(* CODESYS project ExceptionGenerator.library
   TcLibraryId: TE140x Module Vendor|ExceptionGenerator|0.0.0.3
   Company: TE140x Module Vendor
   DefaultNamespace: ExceptionGenerator
   Version: 0.0.0.3
   Placeholder: ExceptionGenerator
   Title: ExceptionGenerator

Project tree, tasks and I/O mapping:
  Version/
    global variables Global_Version
  Pous/
    function block FB_ExceptionGenerator [ST]: FB_exit, FB_init
    TcCOM Wrapper/
      function block FB_ExceptionGenerator_TcCOM_InitStruct [ST]: FB_init, FB_afterinit, Reinit, FB_exit, nTaskOid, nObjectState, ipADI, ipTcComObject, nTaskPriority, nTaskCycleTimeNs, nTaskPort, nTaskSortOrder, eTraceLevelMax, eModuleCaller, eCallerVerification, eStepSizeAdaptation, eExecutionSequence, bExecute, eAccessLockState, eInitExceptionHandling, eUpdateExceptionHandling, stModuleBuildInfo, bInitialized, stInitExceptionInfo, nCycleCount, nExceptionCount, stExeceptionInfo
  Duts/
    data type ST_FB_Main_FB_ExceptionGenerator
    data type ST_FB_exit_FB_ExceptionGenerator
    data type ST_FB_init_FB_ExceptionGenerator
    data type ST_DW_ExceptionGenerator_T
    data type ST_ExtU_ExceptionGenerator_T
    data type ST_ExtY_ExceptionGenerator_T
    data type E_ModuleCaller
    data type E_CallerVerification
    data type E_StepSizeAdaptation
    data type E_ExecutionSequence1
    data type E_FpExcptCtrlSet
    data type ST_FB_ExceptionGenerator_TcCOM_InitStruct
    data type ST_FB_init_FB_ExceptionGenerator_TcCOM_InitStruct
    data type ST_FB_afterinit_FB_ExceptionGenerator_TcCOM_InitStruct
    data type ST_Reinit_FB_ExceptionGenerator_TcCOM_InitStruct
    data type ST_FB_Main_FB_ExceptionGenerator_TcCOM_InitStruct
    data type ST_FB_exit_FB_ExceptionGenerator_TcCOM_InitStruct
    data type ST_GetnTaskOid_FB_ExceptionGenerator_TcCOM_InitStruct
    data type ST_SetnTaskOid_FB_ExceptionGenerator_TcCOM_InitStruct
    data type ST_GetnObjectState_FB_ExceptionGenerator_TcCOM_InitStruct
    data type ST_SetnObjectState_FB_ExceptionGenerator_TcCOM_InitStruct
    data type ST_GetipADI_FB_ExceptionGenerator_TcCOM_InitStruct
    data type ST_SetipADI_FB_ExceptionGenerator_TcCOM_InitStruct
    data type ST_GetipTcComObject_FB_ExceptionGenerator_TcCOM_InitStruct
    data type ST_SetipTcComObject_FB_ExceptionGenerator_TcCOM_InitStruct
    data type ST_ExceptionInfo
    data type ST_ExecutionInfo
    data type ST_GetnTaskPriority_FB_ExceptionGenerator_TcCOM_InitStruct
    data type ST_SetnTaskPriority_FB_ExceptionGenerator_TcCOM_InitStruct
    data type ST_GetnTaskCycleTimeNs_FB_ExceptionGenerator_TcCOM_InitStruct
    data type ST_SetnTaskCycleTimeNs_FB_ExceptionGenerator_TcCOM_InitStruct
    data type ST_GetnTaskPort_FB_ExceptionGenerator_TcCOM_InitStruct
    data type ST_SetnTaskPort_FB_ExceptionGenerator_TcCOM_InitStruct
    data type ST_GetnTaskSortOrder_FB_ExceptionGenerator_TcCOM_InitStruct
    data type ST_SetnTaskSortOrder_FB_ExceptionGenerator_TcCOM_InitStruct
    data type ST_GeteTraceLevelMax_FB_ExceptionGenerator_TcCOM_InitStruct
    data type ST_SeteTraceLevelMax_FB_ExceptionGenerator_TcCOM_InitStruct
    data type ST_GeteModuleCaller_FB_ExceptionGenerator_TcCOM_InitStruct
    data type ST_SeteModuleCaller_FB_ExceptionGenerator_TcCOM_InitStruct
    data type ST_GeteCallerVerification_FB_ExceptionGenerator_TcCOM_InitStruct
    data type ST_SeteCallerVerification_FB_ExceptionGenerator_TcCOM_InitStruct
    data type ST_GeteStepSizeAdaptation_FB_ExceptionGenerator_TcCOM_InitStruct
    data type ST_SeteStepSizeAdaptation_FB_ExceptionGenerator_TcCOM_InitStruct
    data type ST_GeteExecutionSequence_FB_ExceptionGenerator_TcCOM_InitStruct
    data type ST_SeteExecutionSequence_FB_ExceptionGenerator_TcCOM_InitStruct
    data type ST_GetbExecute_FB_ExceptionGenerator_TcCOM_InitStruct
    data type ST_SetbExecute_FB_ExceptionGenerator_TcCOM_InitStruct
    data type ST_GeteAccessLockState_FB_ExceptionGenerator_TcCOM_InitStruct
    data type ST_SeteAccessLockState_FB_ExceptionGenerator_TcCOM_InitStruct
    data type ST_GeteInitExceptionHandling_FB_ExceptionGenerator_TcCOM_InitStruct
    data type ST_SeteInitExceptionHandling_FB_ExceptionGenerator_TcCOM_InitStruct
    data type ST_GeteUpdateExceptionHandling_FB_ExceptionGenerator_TcCOM_InitStruct
    data type ST_SeteUpdateExceptionHandling_FB_ExceptionGenerator_TcCOM_InitStruct
    data type ST_ModuleBuildInfo
    data type ST_GetstModuleBuildInfo_FB_ExceptionGenerator_TcCOM_InitStruct
    data type ST_SetstModuleBuildInfo_FB_ExceptionGenerator_TcCOM_InitStruct
    data type ST_GetbInitialized_FB_ExceptionGenerator_TcCOM_InitStruct
    data type ST_SetbInitialized_FB_ExceptionGenerator_TcCOM_InitStruct
    data type ST_GetstInitExceptionInfo_FB_ExceptionGenerator_TcCOM_InitStruct
    data type ST_SetstInitExceptionInfo_FB_ExceptionGenerator_TcCOM_InitStruct
    data type ST_GetnCycleCount_FB_ExceptionGenerator_TcCOM_InitStruct
    data type ST_SetnCycleCount_FB_ExceptionGenerator_TcCOM_InitStruct
    data type ST_GetnExceptionCount_FB_ExceptionGenerator_TcCOM_InitStruct
    data type ST_SetnExceptionCount_FB_ExceptionGenerator_TcCOM_InitStruct
    data type ST_GetstExeceptionInfo_FB_ExceptionGenerator_TcCOM_InitStruct
    data type ST_SetstExeceptionInfo_FB_ExceptionGenerator_TcCOM_InitStruct
*)

// Duts/ST_FB_Main_FB_ExceptionGenerator

	{attribute 'TcIecLibraryType'}
{attribute 'hide'}
TYPE ST_FB_Main_FB_ExceptionGenerator : 
	STRUCT
		 {attribute 'GUID' := '18071995-0000-0000-0000-000000000018'}
		pInst : PVOID;
		result : BOOL;
		 {attribute 'hide'}
		_reserved1 : UINT_24_56;
	END_STRUCT
END_TYPE

// Duts/ST_FB_exit_FB_ExceptionGenerator

	{attribute 'TcIecLibraryType'}
{attribute 'hide'}
TYPE ST_FB_exit_FB_ExceptionGenerator : 
	STRUCT
		 {attribute 'GUID' := '18071995-0000-0000-0000-000000000018'}
		pInst : PVOID;
		bInCopyCode : BOOL;
		result : BOOL;
		 {attribute 'hide'}
		_reserved1 : UINT_16_48;
	END_STRUCT
END_TYPE

// Duts/ST_FB_init_FB_ExceptionGenerator

	{attribute 'TcIecLibraryType'}
{attribute 'hide'}
TYPE ST_FB_init_FB_ExceptionGenerator : 
	STRUCT
		 {attribute 'GUID' := '18071995-0000-0000-0000-000000000018'}
		pInst : PVOID;
		bInitRetains : BOOL;
		bInCopyCode : BOOL;
		result : BOOL;
		 {attribute 'hide'}
		_reserved1 : UINT_8_40;
	END_STRUCT
END_TYPE

// Duts/ST_DW_ExceptionGenerator_T

	{attribute 'TcIecLibraryType'}
TYPE ST_DW_ExceptionGenerator_T : 
	STRUCT
		fCounter : LREAL;
		fa : LREAL;
		fb : LREAL;
		ffPosInf : LREAL;
		ffNegInf : LREAL;
	END_STRUCT
END_TYPE

// Duts/ST_ExtU_ExceptionGenerator_T

	{attribute 'TcIecLibraryType'}
TYPE ST_ExtU_ExceptionGenerator_T : 
	STRUCT
		bDivByZero : BOOL;
		bFloatingPoint : BOOL;
	END_STRUCT
END_TYPE

// Duts/ST_ExtY_ExceptionGenerator_T

	{attribute 'TcIecLibraryType'}
TYPE ST_ExtY_ExceptionGenerator_T : 
	STRUCT
		fResult : LREAL;
		fCounter : LREAL;
	END_STRUCT
END_TYPE

// Duts/E_ModuleCaller

	{attribute 'TcIecLibraryType'}
TYPE E_ModuleCaller : (
	CyclicTask:=0, 	(* Add to the specified cyclic caller tasks. *)
	Module:=1	(* Don't add to cyclic callers. The module can be called from other TwinCAT modules (e. g. a PLC). *)
) DINT;
END_TYPE

// Duts/E_CallerVerification

	{attribute 'TcIecLibraryType'}
TYPE E_CallerVerification : (
	Default:=0, 	(* Verify the caller task only if the "ModuleCaller" parameter is set to "Module" but not when added to cyclic caller tasks. *)
	Always:=1, 	(* Always verify the caller context to prevent concurrent execution of model code and corresponding DataArea mappings. *)
	Never:=2	(* Skip caller verification to reduce execution times. *)
) DINT;
END_TYPE

// Duts/E_StepSizeAdaptation

	{attribute 'TcIecLibraryType'}
TYPE E_StepSizeAdaptation : (
	RequireMatchingTaskCycleTime:=0, 	(* Don't accept task cycle times other than the Simulink step sizes. *)
	UseTaskCycleTime:=1, 	(* Adapt the Smulink step sizes to the task cycle times. *)
	UseModelStepSize:=2	(* Keep the Smulink step sizes, independent of the callers cycle time. *)
) DINT;
END_TYPE

// Duts/E_ExecutionSequence1

	{attribute 'TcIecLibraryType'}
TYPE E_ExecutionSequence1 : (
	UpdateBeforeOutputMapping:=0, 	(* Input mapping -> State and output update -> Output mapping -> ADS processing *)
	IoAtTaskBegin:=1	(* Input mapping -> Code execution -> Output update -> ADS processing *)
) DINT;
END_TYPE

// Duts/E_FpExcptCtrlSet

	{attribute 'TcIecLibraryType'}
TYPE E_FpExcptCtrlSet : (
	CallerExceptions:=1, 	(* Use the floating point exception settings provided by the caller *)
	ThrowExceptions:=3, 	(* Enable floating point exceptions on invalid operations and divisions by zero *)
	SuppressExceptions:=12, 	(* Disable floating point exceptions. *)
	LogExceptions:=19, 	(* Log exception information. *)
	LogAndHold:=51, 	(* Log exception information and puase execution of the cyclic code after completion of the actual cycle *)
	LogAndCatch:=83, 	(* Log exception information and immediately terminate execution of the cyclic code. Reinitialization is required to restart. *)
	LogAndDump:=147, 	(* Log exception information, create a dump file with detailed exception information and try to continue execution of the cyclic code *)
	LogHoldAndDump:=179, 	(* Log exception information, create a dump file with detailed exception information and puase execution of the cyclic code after completion of the actual cycle *)
	LogCatchAndDump:=211	(* Log exception information, create a dump file with detailed exception information and immediately terminate execution of the cyclic code. Reinitialization is required to restart. *)
) USINT;
END_TYPE

// Duts/ST_FB_ExceptionGenerator_TcCOM_InitStruct

	{attribute 'TcIecLibraryType'}
TYPE ST_FB_ExceptionGenerator_TcCOM_InitStruct : 
	STRUCT
		 {attribute 'GUID' := '18071995-0000-0000-0000-000000000061'}
		eObjState : TCOM_STATE := TCOM_STATE.TCOM_STATE_OP;
		 {attribute 'GUID' := '18071995-0000-0000-0000-00000000000F'}
		nOid : OTCID := 4294967295;
		 {attribute 'GUID' := '18071995-0000-0000-0000-00000000000F'}
		nTaskOid : OTCID;
		{attribute 'hide'}
		nTaskPriority : UDINT;
		{attribute 'hide'}
		nTaskCycleTimeNs : UDINT;
		{attribute 'hide'}
		nTaskPort : UINT;
		 {attribute 'hide'}
		_reserved1 : UINT;
		nTaskSortOrder : UDINT;
		 {attribute 'GUID' := '8007AE3B-86BB-40F2-B385-EF87FCC239A4'}
		eTraceLevelMax : TcTraceLevel := TcTraceLevel.tlInfo;
		eModuleCaller : E_ModuleCaller := E_ModuleCaller.CyclicTask;
		eCallerVerification : E_CallerVerification := E_CallerVerification.Default;
		eStepSizeAdaptation : E_StepSizeAdaptation := E_StepSizeAdaptation.RequireMatchingTaskCycleTime;
		eExecutionSequence : E_ExecutionSequence1 := E_ExecutionSequence1.UpdateBeforeOutputMapping;
		bExecute : BOOL := TRUE;
		 {attribute 'hide'}
		_reserved2 : ARRAY [1..3] OF USINT;
		 {attribute 'GUID' := '18071995-0000-0000-0000-000000000061'}
		eAccessLockState : TCOM_STATE := TCOM_STATE.TCOM_STATE_OP;
		eInitExceptionHandling : E_FpExcptCtrlSet := E_FpExcptCtrlSet.LogCatchAndDump;
		eUpdateExceptionHandling : E_FpExcptCtrlSet := E_FpExcptCtrlSet.LogCatchAndDump;
		 {attribute 'hide'}
		_reserved3 : UINT;
	END_STRUCT
END_TYPE

// Duts/ST_FB_init_FB_ExceptionGenerator_TcCOM_InitStruct

	{attribute 'TcIecLibraryType'}
{attribute 'hide'}
TYPE ST_FB_init_FB_ExceptionGenerator_TcCOM_InitStruct : 
	STRUCT
		 {attribute 'GUID' := '18071995-0000-0000-0000-000000000018'}
		pInst : PVOID;
		bInitRetains : BOOL;
		bInCopyCode : BOOL;
		 {attribute 'hide'}
		_reserved1 : UINT;
		stInit : ST_FB_ExceptionGenerator_TcCOM_InitStruct;
		result : BOOL;
		 {attribute 'hide'}
		_reserved2 : UINT_24_56;
	END_STRUCT
END_TYPE

// Duts/ST_FB_afterinit_FB_ExceptionGenerator_TcCOM_InitStruct

	{attribute 'TcIecLibraryType'}
{attribute 'hide'}
TYPE ST_FB_afterinit_FB_ExceptionGenerator_TcCOM_InitStruct : 
	STRUCT
		 {attribute 'GUID' := '18071995-0000-0000-0000-000000000018'}
		pInst : PVOID;
		result : BOOL;
		 {attribute 'hide'}
		_reserved1 : UINT_24_56;
	END_STRUCT
END_TYPE

// Duts/ST_Reinit_FB_ExceptionGenerator_TcCOM_InitStruct

	{attribute 'TcIecLibraryType'}
{attribute 'hide'}
TYPE ST_Reinit_FB_ExceptionGenerator_TcCOM_InitStruct : 
	STRUCT
		 {attribute 'GUID' := '18071995-0000-0000-0000-000000000018'}
		pInst : PVOID;
		stReInit : ST_FB_ExceptionGenerator_TcCOM_InitStruct;
		result : BOOL;
		 {attribute 'hide'}
		_reserved1 : ARRAY [1..3] OF USINT;
	END_STRUCT
END_TYPE

// Duts/ST_FB_Main_FB_ExceptionGenerator_TcCOM_InitStruct

	{attribute 'TcIecLibraryType'}
{attribute 'hide'}
TYPE ST_FB_Main_FB_ExceptionGenerator_TcCOM_InitStruct : 
	STRUCT
		 {attribute 'GUID' := '18071995-0000-0000-0000-000000000018'}
		pInst : PVOID;
		result : BOOL;
		 {attribute 'hide'}
		_reserved1 : UINT_24_56;
	END_STRUCT
END_TYPE

// Duts/ST_FB_exit_FB_ExceptionGenerator_TcCOM_InitStruct

	{attribute 'TcIecLibraryType'}
{attribute 'hide'}
TYPE ST_FB_exit_FB_ExceptionGenerator_TcCOM_InitStruct : 
	STRUCT
		 {attribute 'GUID' := '18071995-0000-0000-0000-000000000018'}
		pInst : PVOID;
		bInCopyCode : BOOL;
		result : BOOL;
		 {attribute 'hide'}
		_reserved1 : UINT_16_48;
	END_STRUCT
END_TYPE

// Duts/ST_GetnTaskOid_FB_ExceptionGenerator_TcCOM_InitStruct

	{attribute 'TcIecLibraryType'}
{attribute 'hide'}
TYPE ST_GetnTaskOid_FB_ExceptionGenerator_TcCOM_InitStruct : 
	STRUCT
		 {attribute 'GUID' := '18071995-0000-0000-0000-000000000018'}
		pInst : PVOID;
		result : UDINT;
		 {attribute 'hide'}
		_reserved1 : UINT_0_32;
	END_STRUCT
END_TYPE

// Duts/ST_SetnTaskOid_FB_ExceptionGenerator_TcCOM_InitStruct

	{attribute 'TcIecLibraryType'}
{attribute 'hide'}
TYPE ST_SetnTaskOid_FB_ExceptionGenerator_TcCOM_InitStruct : 
	STRUCT
		 {attribute 'GUID' := '18071995-0000-0000-0000-000000000018'}
		pInst : PVOID;
		nParam : UDINT;
		 {attribute 'hide'}
		_reserved1 : UINT_0_32;
	END_STRUCT
END_TYPE

// Duts/ST_GetnObjectState_FB_ExceptionGenerator_TcCOM_InitStruct

	{attribute 'TcIecLibraryType'}
{attribute 'hide'}
TYPE ST_GetnObjectState_FB_ExceptionGenerator_TcCOM_InitStruct : 
	STRUCT
		 {attribute 'GUID' := '18071995-0000-0000-0000-000000000018'}
		pInst : PVOID;
		 {attribute 'GUID' := '18071995-0000-0000-0000-000000000061'}
		result : TCOM_STATE;
		 {attribute 'hide'}
		_reserved1 : UINT_0_32;
	END_STRUCT
END_TYPE

// Duts/ST_SetnObjectState_FB_ExceptionGenerator_TcCOM_InitStruct

	{attribute 'TcIecLibraryType'}
{attribute 'hide'}
TYPE ST_SetnObjectState_FB_ExceptionGenerator_TcCOM_InitStruct : 
	STRUCT
		 {attribute 'GUID' := '18071995-0000-0000-0000-000000000018'}
		pInst : PVOID;
		 {attribute 'GUID' := '18071995-0000-0000-0000-000000000061'}
		eParam : TCOM_STATE;
		 {attribute 'hide'}
		_reserved1 : UINT_0_32;
	END_STRUCT
END_TYPE

// Duts/ST_GetipADI_FB_ExceptionGenerator_TcCOM_InitStruct

	{attribute 'TcIecLibraryType'}
{attribute 'hide'}
TYPE ST_GetipADI_FB_ExceptionGenerator_TcCOM_InitStruct : 
	STRUCT
		 {attribute 'GUID' := '18071995-0000-0000-0000-000000000018'}
		pInst : PVOID;
		 {attribute 'GUID' := '03000012-0000-0000-E000-000000000064'}
		result : ITcADI;
	END_STRUCT
END_TYPE

// Duts/ST_SetipADI_FB_ExceptionGenerator_TcCOM_InitStruct

	{attribute 'TcIecLibraryType'}
{attribute 'hide'}
TYPE ST_SetipADI_FB_ExceptionGenerator_TcCOM_InitStruct : 
	STRUCT
		 {attribute 'GUID' := '18071995-0000-0000-0000-000000000018'}
		pInst : PVOID;
		 {attribute 'GUID' := '03000012-0000-0000-E000-000000000064'}
		ipParam : ITcADI;
	END_STRUCT
END_TYPE

// Duts/ST_GetipTcComObject_FB_ExceptionGenerator_TcCOM_InitStruct

	{attribute 'TcIecLibraryType'}
{attribute 'hide'}
TYPE ST_GetipTcComObject_FB_ExceptionGenerator_TcCOM_InitStruct : 
	STRUCT
		 {attribute 'GUID' := '18071995-0000-0000-0000-000000000018'}
		pInst : PVOID;
		 {attribute 'GUID' := '00000012-0000-0000-E000-000000000064'}
		result : ITComObject;
	END_STRUCT
END_TYPE

// Duts/ST_SetipTcComObject_FB_ExceptionGenerator_TcCOM_InitStruct

	{attribute 'TcIecLibraryType'}
{attribute 'hide'}
TYPE ST_SetipTcComObject_FB_ExceptionGenerator_TcCOM_InitStruct : 
	STRUCT
		 {attribute 'GUID' := '18071995-0000-0000-0000-000000000018'}
		pInst : PVOID;
		 {attribute 'GUID' := '00000012-0000-0000-E000-000000000064'}
		ipParam : ITComObject;
	END_STRUCT
END_TYPE

// Duts/ST_ExceptionInfo

	{attribute 'TcIecLibraryType'}
TYPE ST_ExceptionInfo : 
	STRUCT
		nExceptionCode : DINT;
		 {attribute 'GUID' := '18071995-0000-0000-0000-00010000007F'}
		sTmxName : STRING(127);
		nTmxVersion : UDINT;
		 {attribute 'hide'}
		_reserved1 : ARRAY [1..12] OF USINT;
		nInstructionAddr : UDINT;
		nReturnAddr : UDINT;
		 {attribute 'hide'}
		_reserved2 : ARRAY [1..12] OF USINT;
		bDumpCreated : BOOL;
		 {attribute 'hide'}
		_reserved3 : ARRAY [1..3] OF USINT;
	END_STRUCT
END_TYPE

// Duts/ST_ExecutionInfo

	{attribute 'TcIecLibraryType'}
{attribute 'pack_mode' := '1'}
TYPE ST_ExecutionInfo : 
	STRUCT
		nCycleCount : ULINT;
		nExceptionCount : ULINT;
		stActException : ST_ExceptionInfo;
	END_STRUCT
END_TYPE

// Duts/ST_GetnTaskPriority_FB_ExceptionGenerator_TcCOM_InitStruct

	{attribute 'TcIecLibraryType'}
{attribute 'hide'}
TYPE ST_GetnTaskPriority_FB_ExceptionGenerator_TcCOM_InitStruct : 
	STRUCT
		 {attribute 'GUID' := '18071995-0000-0000-0000-000000000018'}
		pInst : PVOID;
		result : UDINT;
		 {attribute 'hide'}
		_reserved1 : UINT_0_32;
	END_STRUCT
END_TYPE

// Duts/ST_SetnTaskPriority_FB_ExceptionGenerator_TcCOM_InitStruct

	{attribute 'TcIecLibraryType'}
{attribute 'hide'}
TYPE ST_SetnTaskPriority_FB_ExceptionGenerator_TcCOM_InitStruct : 
	STRUCT
		 {attribute 'GUID' := '18071995-0000-0000-0000-000000000018'}
		pInst : PVOID;
		nParam : UDINT;
		 {attribute 'hide'}
		_reserved1 : UINT_0_32;
	END_STRUCT
END_TYPE

// Duts/ST_GetnTaskCycleTimeNs_FB_ExceptionGenerator_TcCOM_InitStruct

	{attribute 'TcIecLibraryType'}
{attribute 'hide'}
TYPE ST_GetnTaskCycleTimeNs_FB_ExceptionGenerator_TcCOM_InitStruct : 
	STRUCT
		 {attribute 'GUID' := '18071995-0000-0000-0000-000000000018'}
		pInst : PVOID;
		result : UDINT;
		 {attribute 'hide'}
		_reserved1 : UINT_0_32;
	END_STRUCT
END_TYPE

// Duts/ST_SetnTaskCycleTimeNs_FB_ExceptionGenerator_TcCOM_InitStruct

	{attribute 'TcIecLibraryType'}
{attribute 'hide'}
TYPE ST_SetnTaskCycleTimeNs_FB_ExceptionGenerator_TcCOM_InitStruct : 
	STRUCT
		 {attribute 'GUID' := '18071995-0000-0000-0000-000000000018'}
		pInst : PVOID;
		nParam : UDINT;
		 {attribute 'hide'}
		_reserved1 : UINT_0_32;
	END_STRUCT
END_TYPE

// Duts/ST_GetnTaskPort_FB_ExceptionGenerator_TcCOM_InitStruct

	{attribute 'TcIecLibraryType'}
{attribute 'hide'}
TYPE ST_GetnTaskPort_FB_ExceptionGenerator_TcCOM_InitStruct : 
	STRUCT
		 {attribute 'GUID' := '18071995-0000-0000-0000-000000000018'}
		pInst : PVOID;
		result : UINT;
		 {attribute 'hide'}
		_reserved1 : UINT_16_48;
	END_STRUCT
END_TYPE

// Duts/ST_SetnTaskPort_FB_ExceptionGenerator_TcCOM_InitStruct

	{attribute 'TcIecLibraryType'}
{attribute 'hide'}
TYPE ST_SetnTaskPort_FB_ExceptionGenerator_TcCOM_InitStruct : 
	STRUCT
		 {attribute 'GUID' := '18071995-0000-0000-0000-000000000018'}
		pInst : PVOID;
		nParam : UINT;
		 {attribute 'hide'}
		_reserved1 : UINT_16_48;
	END_STRUCT
END_TYPE

// Duts/ST_GetnTaskSortOrder_FB_ExceptionGenerator_TcCOM_InitStruct

	{attribute 'TcIecLibraryType'}
{attribute 'hide'}
TYPE ST_GetnTaskSortOrder_FB_ExceptionGenerator_TcCOM_InitStruct : 
	STRUCT
		 {attribute 'GUID' := '18071995-0000-0000-0000-000000000018'}
		pInst : PVOID;
		result : UDINT;
		 {attribute 'hide'}
		_reserved1 : UINT_0_32;
	END_STRUCT
END_TYPE

// Duts/ST_SetnTaskSortOrder_FB_ExceptionGenerator_TcCOM_InitStruct

	{attribute 'TcIecLibraryType'}
{attribute 'hide'}
TYPE ST_SetnTaskSortOrder_FB_ExceptionGenerator_TcCOM_InitStruct : 
	STRUCT
		 {attribute 'GUID' := '18071995-0000-0000-0000-000000000018'}
		pInst : PVOID;
		nParam : UDINT;
		 {attribute 'hide'}
		_reserved1 : UINT_0_32;
	END_STRUCT
END_TYPE

// Duts/ST_GeteTraceLevelMax_FB_ExceptionGenerator_TcCOM_InitStruct

	{attribute 'TcIecLibraryType'}
{attribute 'hide'}
TYPE ST_GeteTraceLevelMax_FB_ExceptionGenerator_TcCOM_InitStruct : 
	STRUCT
		 {attribute 'GUID' := '18071995-0000-0000-0000-000000000018'}
		pInst : PVOID;
		 {attribute 'GUID' := '8007AE3B-86BB-40F2-B385-EF87FCC239A4'}
		result : TcTraceLevel;
		 {attribute 'hide'}
		_reserved1 : UINT_0_32;
	END_STRUCT
END_TYPE

// Duts/ST_SeteTraceLevelMax_FB_ExceptionGenerator_TcCOM_InitStruct

	{attribute 'TcIecLibraryType'}
{attribute 'hide'}
TYPE ST_SeteTraceLevelMax_FB_ExceptionGenerator_TcCOM_InitStruct : 
	STRUCT
		 {attribute 'GUID' := '18071995-0000-0000-0000-000000000018'}
		pInst : PVOID;
		 {attribute 'GUID' := '8007AE3B-86BB-40F2-B385-EF87FCC239A4'}
		eParam : TcTraceLevel;
		 {attribute 'hide'}
		_reserved1 : UINT_0_32;
	END_STRUCT
END_TYPE

// Duts/ST_GeteModuleCaller_FB_ExceptionGenerator_TcCOM_InitStruct

	{attribute 'TcIecLibraryType'}
{attribute 'hide'}
TYPE ST_GeteModuleCaller_FB_ExceptionGenerator_TcCOM_InitStruct : 
	STRUCT
		 {attribute 'GUID' := '18071995-0000-0000-0000-000000000018'}
		pInst : PVOID;
		result : E_ModuleCaller;
		 {attribute 'hide'}
		_reserved1 : UINT_0_32;
	END_STRUCT
END_TYPE

// Duts/ST_SeteModuleCaller_FB_ExceptionGenerator_TcCOM_InitStruct

	{attribute 'TcIecLibraryType'}
{attribute 'hide'}
TYPE ST_SeteModuleCaller_FB_ExceptionGenerator_TcCOM_InitStruct : 
	STRUCT
		 {attribute 'GUID' := '18071995-0000-0000-0000-000000000018'}
		pInst : PVOID;
		eParam : E_ModuleCaller;
		 {attribute 'hide'}
		_reserved1 : UINT_0_32;
	END_STRUCT
END_TYPE

// Duts/ST_GeteCallerVerification_FB_ExceptionGenerator_TcCOM_InitStruct

	{attribute 'TcIecLibraryType'}
{attribute 'hide'}
TYPE ST_GeteCallerVerification_FB_ExceptionGenerator_TcCOM_InitStruct : 
	STRUCT
		 {attribute 'GUID' := '18071995-0000-0000-0000-000000000018'}
		pInst : PVOID;
		result : E_CallerVerification;
		 {attribute 'hide'}
		_reserved1 : UINT_0_32;
	END_STRUCT
END_TYPE

// Duts/ST_SeteCallerVerification_FB_ExceptionGenerator_TcCOM_InitStruct

	{attribute 'TcIecLibraryType'}
{attribute 'hide'}
TYPE ST_SeteCallerVerification_FB_ExceptionGenerator_TcCOM_InitStruct : 
	STRUCT
		 {attribute 'GUID' := '18071995-0000-0000-0000-000000000018'}
		pInst : PVOID;
		eParam : E_CallerVerification;
		 {attribute 'hide'}
		_reserved1 : UINT_0_32;
	END_STRUCT
END_TYPE

// Duts/ST_GeteStepSizeAdaptation_FB_ExceptionGenerator_TcCOM_InitStruct

	{attribute 'TcIecLibraryType'}
{attribute 'hide'}
TYPE ST_GeteStepSizeAdaptation_FB_ExceptionGenerator_TcCOM_InitStruct : 
	STRUCT
		 {attribute 'GUID' := '18071995-0000-0000-0000-000000000018'}
		pInst : PVOID;
		result : E_StepSizeAdaptation;
		 {attribute 'hide'}
		_reserved1 : UINT_0_32;
	END_STRUCT
END_TYPE

// Duts/ST_SeteStepSizeAdaptation_FB_ExceptionGenerator_TcCOM_InitStruct

	{attribute 'TcIecLibraryType'}
{attribute 'hide'}
TYPE ST_SeteStepSizeAdaptation_FB_ExceptionGenerator_TcCOM_InitStruct : 
	STRUCT
		 {attribute 'GUID' := '18071995-0000-0000-0000-000000000018'}
		pInst : PVOID;
		eParam : E_StepSizeAdaptation;
		 {attribute 'hide'}
		_reserved1 : UINT_0_32;
	END_STRUCT
END_TYPE

// Duts/ST_GeteExecutionSequence_FB_ExceptionGenerator_TcCOM_InitStruct

	{attribute 'TcIecLibraryType'}
{attribute 'hide'}
TYPE ST_GeteExecutionSequence_FB_ExceptionGenerator_TcCOM_InitStruct : 
	STRUCT
		 {attribute 'GUID' := '18071995-0000-0000-0000-000000000018'}
		pInst : PVOID;
		result : E_ExecutionSequence1;
		 {attribute 'hide'}
		_reserved1 : UINT_0_32;
	END_STRUCT
END_TYPE

// Duts/ST_SeteExecutionSequence_FB_ExceptionGenerator_TcCOM_InitStruct

	{attribute 'TcIecLibraryType'}
{attribute 'hide'}
TYPE ST_SeteExecutionSequence_FB_ExceptionGenerator_TcCOM_InitStruct : 
	STRUCT
		 {attribute 'GUID' := '18071995-0000-0000-0000-000000000018'}
		pInst : PVOID;
		eParam : E_ExecutionSequence1;
		 {attribute 'hide'}
		_reserved1 : UINT_0_32;
	END_STRUCT
END_TYPE

// Duts/ST_GetbExecute_FB_ExceptionGenerator_TcCOM_InitStruct

	{attribute 'TcIecLibraryType'}
{attribute 'hide'}
TYPE ST_GetbExecute_FB_ExceptionGenerator_TcCOM_InitStruct : 
	STRUCT
		 {attribute 'GUID' := '18071995-0000-0000-0000-000000000018'}
		pInst : PVOID;
		result : BOOL;
		 {attribute 'hide'}
		_reserved1 : UINT_24_56;
	END_STRUCT
END_TYPE

// Duts/ST_SetbExecute_FB_ExceptionGenerator_TcCOM_InitStruct

	{attribute 'TcIecLibraryType'}
{attribute 'hide'}
TYPE ST_SetbExecute_FB_ExceptionGenerator_TcCOM_InitStruct : 
	STRUCT
		 {attribute 'GUID' := '18071995-0000-0000-0000-000000000018'}
		pInst : PVOID;
		bParam : BOOL;
		 {attribute 'hide'}
		_reserved1 : UINT_24_56;
	END_STRUCT
END_TYPE

// Duts/ST_GeteAccessLockState_FB_ExceptionGenerator_TcCOM_InitStruct

	{attribute 'TcIecLibraryType'}
{attribute 'hide'}
TYPE ST_GeteAccessLockState_FB_ExceptionGenerator_TcCOM_InitStruct : 
	STRUCT
		 {attribute 'GUID' := '18071995-0000-0000-0000-000000000018'}
		pInst : PVOID;
		 {attribute 'GUID' := '18071995-0000-0000-0000-000000000061'}
		result : TCOM_STATE;
		 {attribute 'hide'}
		_reserved1 : UINT_0_32;
	END_STRUCT
END_TYPE

// Duts/ST_SeteAccessLockState_FB_ExceptionGenerator_TcCOM_InitStruct

	{attribute 'TcIecLibraryType'}
{attribute 'hide'}
TYPE ST_SeteAccessLockState_FB_ExceptionGenerator_TcCOM_InitStruct : 
	STRUCT
		 {attribute 'GUID' := '18071995-0000-0000-0000-000000000018'}
		pInst : PVOID;
		 {attribute 'GUID' := '18071995-0000-0000-0000-000000000061'}
		eParam : TCOM_STATE;
		 {attribute 'hide'}
		_reserved1 : UINT_0_32;
	END_STRUCT
END_TYPE

// Duts/ST_GeteInitExceptionHandling_FB_ExceptionGenerator_TcCOM_InitStruct

	{attribute 'TcIecLibraryType'}
{attribute 'hide'}
TYPE ST_GeteInitExceptionHandling_FB_ExceptionGenerator_TcCOM_InitStruct : 
	STRUCT
		 {attribute 'GUID' := '18071995-0000-0000-0000-000000000018'}
		pInst : PVOID;
		result : E_FpExcptCtrlSet;
		 {attribute 'hide'}
		_reserved1 : UINT_24_56;
	END_STRUCT
END_TYPE

// Duts/ST_SeteInitExceptionHandling_FB_ExceptionGenerator_TcCOM_InitStruct

	{attribute 'TcIecLibraryType'}
{attribute 'hide'}
TYPE ST_SeteInitExceptionHandling_FB_ExceptionGenerator_TcCOM_InitStruct : 
	STRUCT
		 {attribute 'GUID' := '18071995-0000-0000-0000-000000000018'}
		pInst : PVOID;
		eParam : E_FpExcptCtrlSet;
		 {attribute 'hide'}
		_reserved1 : UINT_24_56;
	END_STRUCT
END_TYPE

// Duts/ST_GeteUpdateExceptionHandling_FB_ExceptionGenerator_TcCOM_InitStruct

	{attribute 'TcIecLibraryType'}
{attribute 'hide'}
TYPE ST_GeteUpdateExceptionHandling_FB_ExceptionGenerator_TcCOM_InitStruct : 
	STRUCT
		 {attribute 'GUID' := '18071995-0000-0000-0000-000000000018'}
		pInst : PVOID;
		result : E_FpExcptCtrlSet;
		 {attribute 'hide'}
		_reserved1 : UINT_24_56;
	END_STRUCT
END_TYPE

// Duts/ST_SeteUpdateExceptionHandling_FB_ExceptionGenerator_TcCOM_InitStruct

	{attribute 'TcIecLibraryType'}
{attribute 'hide'}
TYPE ST_SeteUpdateExceptionHandling_FB_ExceptionGenerator_TcCOM_InitStruct : 
	STRUCT
		 {attribute 'GUID' := '18071995-0000-0000-0000-000000000018'}
		pInst : PVOID;
		eParam : E_FpExcptCtrlSet;
		 {attribute 'hide'}
		_reserved1 : UINT_24_56;
	END_STRUCT
END_TYPE

// Duts/ST_ModuleBuildInfo

	{attribute 'TcIecLibraryType'}
TYPE ST_ModuleBuildInfo : 
	STRUCT
		nTcBuild : UDINT;
		nTcRevision : UDINT;
		bDebug : BOOL;
		 {attribute 'hide'}
		_reserved1 : ARRAY [1..3] OF USINT;
	END_STRUCT
END_TYPE

// Duts/ST_GetstModuleBuildInfo_FB_ExceptionGenerator_TcCOM_InitStruct

	{attribute 'TcIecLibraryType'}
{attribute 'hide'}
TYPE ST_GetstModuleBuildInfo_FB_ExceptionGenerator_TcCOM_InitStruct : 
	STRUCT
		 {attribute 'GUID' := '18071995-0000-0000-0000-000000000018'}
		pInst : PVOID;
		result : ST_ModuleBuildInfo;
		 {attribute 'hide'}
		_reserved1 : UINT_0_32;
	END_STRUCT
END_TYPE

// Duts/ST_SetstModuleBuildInfo_FB_ExceptionGenerator_TcCOM_InitStruct

	{attribute 'TcIecLibraryType'}
{attribute 'hide'}
TYPE ST_SetstModuleBuildInfo_FB_ExceptionGenerator_TcCOM_InitStruct : 
	STRUCT
		 {attribute 'GUID' := '18071995-0000-0000-0000-000000000018'}
		pInst : PVOID;
		stParam : ST_ModuleBuildInfo;
		 {attribute 'hide'}
		_reserved1 : UINT_0_32;
	END_STRUCT
END_TYPE

// Duts/ST_GetbInitialized_FB_ExceptionGenerator_TcCOM_InitStruct

	{attribute 'TcIecLibraryType'}
{attribute 'hide'}
TYPE ST_GetbInitialized_FB_ExceptionGenerator_TcCOM_InitStruct : 
	STRUCT
		 {attribute 'GUID' := '18071995-0000-0000-0000-000000000018'}
		pInst : PVOID;
		result : BOOL;
		 {attribute 'hide'}
		_reserved1 : UINT_24_56;
	END_STRUCT
END_TYPE

// Duts/ST_SetbInitialized_FB_ExceptionGenerator_TcCOM_InitStruct

	{attribute 'TcIecLibraryType'}
{attribute 'hide'}
TYPE ST_SetbInitialized_FB_ExceptionGenerator_TcCOM_InitStruct : 
	STRUCT
		 {attribute 'GUID' := '18071995-0000-0000-0000-000000000018'}
		pInst : PVOID;
		bParam : BOOL;
		 {attribute 'hide'}
		_reserved1 : UINT_24_56;
	END_STRUCT
END_TYPE

// Duts/ST_GetstInitExceptionInfo_FB_ExceptionGenerator_TcCOM_InitStruct

	{attribute 'TcIecLibraryType'}
{attribute 'hide'}
TYPE ST_GetstInitExceptionInfo_FB_ExceptionGenerator_TcCOM_InitStruct : 
	STRUCT
		 {attribute 'GUID' := '18071995-0000-0000-0000-000000000018'}
		pInst : PVOID;
		result : ST_ExceptionInfo;
		 {attribute 'hide'}
		_reserved1 : UINT_0_32;
	END_STRUCT
END_TYPE

// Duts/ST_SetstInitExceptionInfo_FB_ExceptionGenerator_TcCOM_InitStruct

	{attribute 'TcIecLibraryType'}
{attribute 'hide'}
TYPE ST_SetstInitExceptionInfo_FB_ExceptionGenerator_TcCOM_InitStruct : 
	STRUCT
		 {attribute 'GUID' := '18071995-0000-0000-0000-000000000018'}
		pInst : PVOID;
		stParam : ST_ExceptionInfo;
		 {attribute 'hide'}
		_reserved1 : UINT_0_32;
	END_STRUCT
END_TYPE

// Duts/ST_GetnCycleCount_FB_ExceptionGenerator_TcCOM_InitStruct

	{attribute 'TcIecLibraryType'}
{attribute 'hide'}
TYPE ST_GetnCycleCount_FB_ExceptionGenerator_TcCOM_InitStruct : 
	STRUCT
		 {attribute 'GUID' := '18071995-0000-0000-0000-000000000018'}
		pInst : PVOID;
		result : ULINT;
	END_STRUCT
END_TYPE

// Duts/ST_SetnCycleCount_FB_ExceptionGenerator_TcCOM_InitStruct

	{attribute 'TcIecLibraryType'}
{attribute 'hide'}
TYPE ST_SetnCycleCount_FB_ExceptionGenerator_TcCOM_InitStruct : 
	STRUCT
		 {attribute 'GUID' := '18071995-0000-0000-0000-000000000018'}
		pInst : PVOID;
		nParam : ULINT;
	END_STRUCT
END_TYPE

// Duts/ST_GetnExceptionCount_FB_ExceptionGenerator_TcCOM_InitStruct

	{attribute 'TcIecLibraryType'}
{attribute 'hide'}
TYPE ST_GetnExceptionCount_FB_ExceptionGenerator_TcCOM_InitStruct : 
	STRUCT
		 {attribute 'GUID' := '18071995-0000-0000-0000-000000000018'}
		pInst : PVOID;
		result : ULINT;
	END_STRUCT
END_TYPE

// Duts/ST_SetnExceptionCount_FB_ExceptionGenerator_TcCOM_InitStruct

	{attribute 'TcIecLibraryType'}
{attribute 'hide'}
TYPE ST_SetnExceptionCount_FB_ExceptionGenerator_TcCOM_InitStruct : 
	STRUCT
		 {attribute 'GUID' := '18071995-0000-0000-0000-000000000018'}
		pInst : PVOID;
		nParam : ULINT;
	END_STRUCT
END_TYPE

// Duts/ST_GetstExeceptionInfo_FB_ExceptionGenerator_TcCOM_InitStruct

	{attribute 'TcIecLibraryType'}
{attribute 'hide'}
TYPE ST_GetstExeceptionInfo_FB_ExceptionGenerator_TcCOM_InitStruct : 
	STRUCT
		 {attribute 'GUID' := '18071995-0000-0000-0000-000000000018'}
		pInst : PVOID;
		result : ST_ExceptionInfo;
		 {attribute 'hide'}
		_reserved1 : UINT_0_32;
	END_STRUCT
END_TYPE

// Duts/ST_SetstExeceptionInfo_FB_ExceptionGenerator_TcCOM_InitStruct

	{attribute 'TcIecLibraryType'}
{attribute 'hide'}
TYPE ST_SetstExeceptionInfo_FB_ExceptionGenerator_TcCOM_InitStruct : 
	STRUCT
		 {attribute 'GUID' := '18071995-0000-0000-0000-000000000018'}
		pInst : PVOID;
		stParam : ST_ExceptionInfo;
		 {attribute 'hide'}
		_reserved1 : UINT_0_32;
	END_STRUCT
END_TYPE

// Version/Global_Version
{attribute 'TcGenerated'}
// This function has been automatically generated from the project information.
VAR_GLOBAL CONSTANT
	{attribute 'const_non_replaced'}
	{attribute 'linkalways'}
	stLibVersion_ExceptionGenerator : ST_LibVersion := (iMajor := 0, iMinor := 0, iBuild := 0, iRevision := 3, sVersion := '0.0.0.3');
	{attribute 'const_non_replaced'}
	{attribute 'linkalways'}
	sLibraryId_ExceptionGenerator : String := 'TE140x Module Vendor|ExceptionGenerator|0.0.0.3';
END_VAR

// Pous/FB_ExceptionGenerator

	{attribute 'c++_compatible'}
	{attribute 'external_name' := 'FB_ExceptionGenerator_GUID_4212010D_4B68_476E_4700_4FD61F16D02E'}
	{attribute 'TcIecLibraryType'}
	FUNCTION_BLOCK FB_ExceptionGenerator
	VAR
		{attribute 'hide'}
		{attribute 'no_copy'}
		 {attribute 'GUID' := '18071995-0000-0000-0000-000000000018'}
		_internal_data : PVOID;
	END_VAR
	VAR_INPUT
		bDivByZero : BOOL;
		bFloatingPoint : BOOL;
	END_VAR
	VAR
		 {attribute 'hide'}
		_reserved1 : ARRAY [1..6] OF USINT;
	END_VAR
	VAR_OUTPUT
		fResult : LREAL;
		fCounter : LREAL;
	END_VAR
	VAR
		 {attribute 'GUID' := '18071995-0000-0000-0000-000000000018'}
		pExceptionGenerator_Obj : PVOID;
	END_VAR


	METHOD FB_exit : BOOL
	VAR_INPUT
		bInCopyCode : BOOL;
	END_VAR
END_METHOD


	METHOD FB_init : BOOL
	VAR_INPUT
		bInitRetains : BOOL;
		bInCopyCode : BOOL;
	END_VAR
END_METHOD

END_FUNCTION_BLOCK

// Pous/TcCOM Wrapper/FB_ExceptionGenerator_TcCOM_InitStruct

	{attribute 'c++_compatible'}
	{attribute 'pack_mode' := '1'}
	{attribute 'external_name' := 'FB_ExceptionGenerator_TcCOM_InitStruct_GUID_BBE507A2_AE29_AD46_CE6E_88F8705D8E6E'}
	{attribute 'TcIecLibraryType'}
	{attribute 'call_after_init'}
	FUNCTION_BLOCK FB_ExceptionGenerator_TcCOM_InitStruct
	VAR
		{attribute 'hide'}
		{attribute 'no_copy'}
		 {attribute 'GUID' := '18071995-0000-0000-0000-000000000018'}
		p_internal_ : PVOID;
	END_VAR
	VAR_INPUT
		stExceptionGenerator_U : ST_ExtU_ExceptionGenerator_T;
	END_VAR
	VAR
		 {attribute 'hide'}
		_reserved1 : ARRAY [1..6] OF USINT;
	END_VAR
	VAR_OUTPUT
		stExceptionGenerator_Y : ST_ExtY_ExceptionGenerator_T;
		stExecutionInfo : ST_ExecutionInfo;
	END_VAR
	VAR
		 {attribute 'hide'}
		_reserved2 : UINT_0_32;
		pExceptionGenerator_U : POINTER TO ST_ExtU_ExceptionGenerator_T;
		pExceptionGenerator_Y : POINTER TO ST_ExtY_ExceptionGenerator_T;
		pExecutionInfo : POINTER TO ST_ExecutionInfo;
		 {attribute 'GUID' := '00000001-0000-0000-E000-000000000064'}
		ipITcUnknown : ITcUnknown;
		 {attribute 'GUID' := '00000002-0000-0000-E000-000000000064'}
		ipITcPersist : ITcPersist;
		 {attribute 'GUID' := '00000012-0000-0000-E000-000000000064'}
		ipITComObject : ITComObject;
		 {attribute 'GUID' := '03000018-0000-0000-E000-000000000064'}
		ipITcWatchSource : ITcWatchSource;
		 {attribute 'GUID' := '03000010-0000-0000-E000-000000000064'}
		ipITcCyclic : ITcCyclic;
		 {attribute 'GUID' := '03000025-0000-0000-E000-000000000064'}
		ipITcPostCyclic : ITcPostCyclic;
		 {attribute 'GUID' := '03000012-0000-0000-E000-000000000064'}
		ipITcADI : ITcADI;
		stInit : ST_FB_ExceptionGenerator_TcCOM_InitStruct;
		 {attribute 'hide'}
		_reserved3 : UINT_0_32;
	END_VAR


	METHOD FB_init : BOOL
	VAR_INPUT
		bInitRetains : BOOL;
		bInCopyCode : BOOL;
 {attribute 'GUID' := 'BC556B36-5112-E529-3509-4590C3374233'}
				stInit : ST_FB_ExceptionGenerator_TcCOM_InitStruct;
	END_VAR
END_METHOD


	{attribute 'call_after_init'}
	METHOD FB_afterinit : BOOL
END_METHOD


	METHOD Reinit : BOOL
	VAR_INPUT
 {attribute 'GUID' := 'BC556B36-5112-E529-3509-4590C3374233'}
				stReInit : ST_FB_ExceptionGenerator_TcCOM_InitStruct;
	END_VAR
END_METHOD


	METHOD FB_exit : BOOL
	VAR_INPUT
		bInCopyCode : BOOL;
	END_VAR
END_METHOD


	PROPERTY nTaskOid : UDINT
SET
END_SET
GET
END_GET
END_PROPERTY


	PROPERTY nObjectState : TCOM_STATE
SET
END_SET
GET
END_GET
END_PROPERTY


	PROPERTY ipADI : ITcADI
SET
END_SET
GET
END_GET
END_PROPERTY


	PROPERTY ipTcComObject : ITComObject
SET
END_SET
GET
END_GET
END_PROPERTY


{attribute 'monitoring' := 'call'}
	PROPERTY nTaskPriority : UDINT
SET
END_SET
GET
END_GET
END_PROPERTY


{attribute 'monitoring' := 'call'}
	PROPERTY nTaskCycleTimeNs : UDINT
SET
END_SET
GET
END_GET
END_PROPERTY


{attribute 'monitoring' := 'call'}
	PROPERTY nTaskPort : UINT
SET
END_SET
GET
END_GET
END_PROPERTY


{attribute 'monitoring' := 'call'}
	PROPERTY nTaskSortOrder : UDINT
SET
END_SET
GET
END_GET
END_PROPERTY


{attribute 'monitoring' := 'call'}
	PROPERTY eTraceLevelMax : TcTraceLevel
SET
END_SET
GET
END_GET
END_PROPERTY


{attribute 'monitoring' := 'call'}
	PROPERTY eModuleCaller : ModuleCaller
SET
END_SET
GET
END_GET
END_PROPERTY


{attribute 'monitoring' := 'call'}
	PROPERTY eCallerVerification : CallerVerification
SET
END_SET
GET
END_GET
END_PROPERTY


{attribute 'monitoring' := 'call'}
	PROPERTY eStepSizeAdaptation : StepSizeAdaptation
SET
END_SET
GET
END_GET
END_PROPERTY


{attribute 'monitoring' := 'call'}
	PROPERTY eExecutionSequence : ExecutionSequence1
SET
END_SET
GET
END_GET
END_PROPERTY


{attribute 'monitoring' := 'call'}
	PROPERTY bExecute : BOOL
SET
END_SET
GET
END_GET
END_PROPERTY


{attribute 'monitoring' := 'call'}
	PROPERTY eAccessLockState : TCOM_STATE
SET
END_SET
GET
END_GET
END_PROPERTY


{attribute 'monitoring' := 'call'}
	PROPERTY eInitExceptionHandling : FpExcptCtrlSet
SET
END_SET
GET
END_GET
END_PROPERTY


{attribute 'monitoring' := 'call'}
	PROPERTY eUpdateExceptionHandling : FpExcptCtrlSet
SET
END_SET
GET
END_GET
END_PROPERTY


{attribute 'monitoring' := 'variable'}
	PROPERTY stModuleBuildInfo : ModuleBuildInfo
SET
END_SET
GET
END_GET
END_PROPERTY


{attribute 'monitoring' := 'call'}
	PROPERTY bInitialized : BOOL
SET
END_SET
GET
END_GET
END_PROPERTY


{attribute 'monitoring' := 'variable'}
	PROPERTY stInitExceptionInfo : ExceptionInfo
SET
END_SET
GET
END_GET
END_PROPERTY


{attribute 'monitoring' := 'call'}
	PROPERTY nCycleCount : ULINT
SET
END_SET
GET
END_GET
END_PROPERTY


{attribute 'monitoring' := 'call'}
	PROPERTY nExceptionCount : ULINT
SET
END_SET
GET
END_GET
END_PROPERTY


{attribute 'monitoring' := 'variable'}
	PROPERTY stExeceptionInfo : ExceptionInfo
SET
END_SET
GET
END_GET
END_PROPERTY

END_FUNCTION_BLOCK
